# EPICS autosave request: SIS8300bpmApp/Db/SIS8300bpmN_settings.req
$(P)$(R)ConvFactor
